(* Logix 5000 project; controller test vendor 1 type 14 code 196 rev 35.11; software revision 35.00 *)

TASK MainTask (continuous, watchdog 500 ms) : MainProgram

MODULES
   Local : vendor 1 type 14 code 196 (5069 0, rev 35.11)
END_MODULES

ADD_ON_INSTRUCTION Casting_Process   (* revision 1.0 *)
VAR_OUTPUT
   Header_Left : BOOL; {access Read Only, visible}
END_VAR
VAR_INPUT
   BW_Limit : BOOL; {required}
   Header_FW : BOOL; {required}
END_VAR
VAR_OUTPUT
   Casting : BOOL; {visible}
   Casting_Done : BOOL; {access Read Only, visible}
END_VAR
VAR
   Timer : TIMER := (PRE := 1500); {access None}
   Timer_1 : TIMER := (PRE := 2000); {access None}
END_VAR

ROUTINE Logic   (* ladder *)
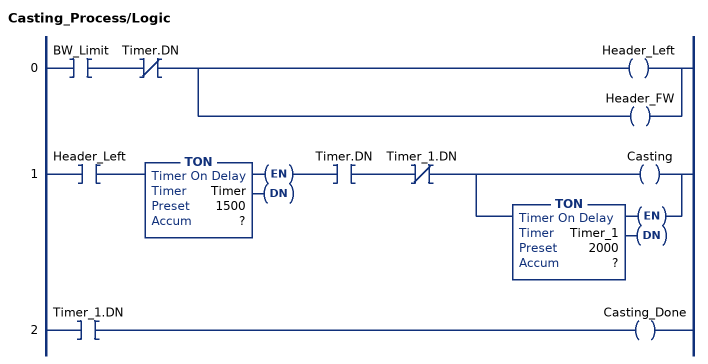
   0: XIC(BW_Limit)XIO(Timer.DN)[OTE(Header_Left) ,OTE(Header_FW) ];
   1: XIC(Header_Left)TON(Timer,?,?)XIC(Timer.DN)XIO(Timer_1.DN)[OTE(Casting) ,TON(Timer_1,?,?) ];
   2: XIC(Timer_1.DN)OTE(Casting_Done);
END_ROUTINE
END_ADD_ON_INSTRUCTION

ADD_ON_INSTRUCTION Molds_Tem   (* revision 1.0 *)
VAR_INPUT
   Temperature : REAL; {required}
END_VAR
VAR_OUTPUT
   Heating : BOOL; {access Read Only, visible}
   R : BOOL; {access Read Only, visible}
END_VAR

ROUTINE Logic   (* ladder *)
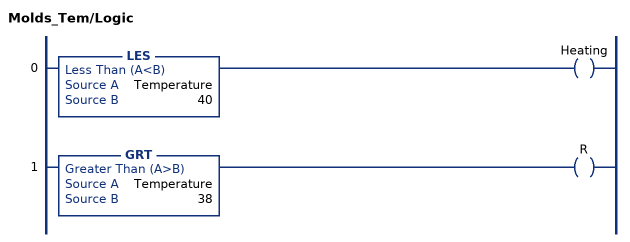
   0: LES(Temperature,40)OTE(Heating);
   1: GRT(Temperature,38)OTE(R);
END_ROUTINE
END_ADD_ON_INSTRUCTION

PROGRAM MainProgram   (* main routine MainRoutine *)
VAR
   Air_Valv : BOOL;
   BW_Limit : BOOL[32];
   Car_BW : BOOL;
   Car_Forward : BOOL;
   Car_FW : BOOL;
   Carriage : BOOL;
   Casting_Process_1 : Casting_Process;
   Casting_Process_2 : Casting_Process;
   Casting_Process_3 : Casting_Process;
   Casting_Process_4 : Casting_Process;
   Casting_Process_5 : Casting_Process;
   Casting_Process_6 : Casting_Process;
   Casting_Process_7 : Casting_Process;
   Casting_Process_8 : Casting_Process;
   Chem_Valv : BOOL;
   Emergency_Button : BOOL;
   Front_Limit : BOOL;
   FW_Limit : BOOL;
   Header_BW : BOOL;
   Header_FW : BOOL[32];
   Header_Right : BOOL;
   Initial_Position : BOOL;
   Light_Auto : BOOL;   // Automatic Light
   Light_Emer : BOOL;
   Light_Man : BOOL;   // Manual Light
   Manual : DINT;
   MTem_1 : Molds_Tem;
   MTem_2 : Molds_Tem;
   MTem_3 : Molds_Tem;
   MTem_4 : Molds_Tem;
   MTem_5 : Molds_Tem;
   MTem_6 : Molds_Tem;
   MTem_7 : Molds_Tem;
   MTem_8 : Molds_Tem;
   PB_AutoMan : BOOL;
   PB_Pouring_Material : BOOL;
   PB_Turn_Table : BOOL;
   PB_Valve_Air : BOOL;
   PB_Valve_Chemical : BOOL;
   Pouring_Material : BOOL;
   Preset_Time : DINT;
   Process_Auto : DINT;
   Process_Station : DINT;
   Ready : BOOL;
   Solenoid_with_chemical : BOOL;
   Solenoid_with_compressed_air : BOOL;
   Start_Button : BOOL;
   Strain : BOOL;
   Switch_Car_BW : BOOL;
   Switch_Car_Forward : BOOL;
   Switch_Header_BW : BOOL;
   Switch_Header_FW : BOOL;
   Tem_1 : REAL;
   Tem_2 : REAL;
   Tem_3 : REAL;
   Tem_4 : REAL;
   Tem_5 : REAL;
   Tem_6 : REAL;
   Tem_7 : REAL;
   Tem_8 : REAL;
   Tem_Ready : BOOL;
   Time_Air_Valv : TIMER := (PRE := 3000);
   Time_Chem_Valv : TIMER := (PRE := 1000);
   Time_Strain : DINT;
   Timer_1 : TIMER := (PRE := 10000);
   Timer_2 : TIMER := (PRE := 1500);
   Turn_Table : BOOL;
END_VAR

ROUTINE Automatic   (* ladder *)
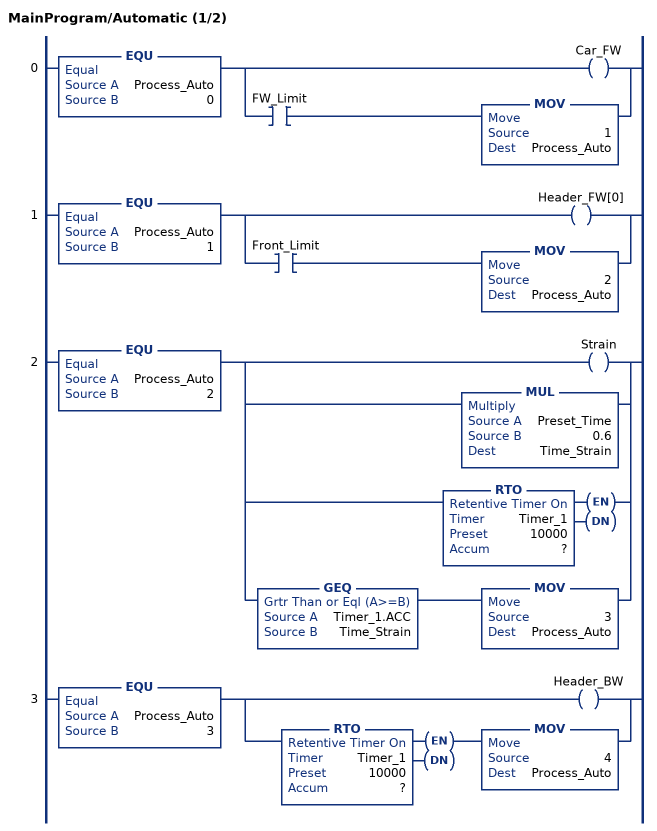
   0: EQU(Process_Auto,0)[OTE(Car_FW) ,XIC(FW_Limit) MOV(1,Process_Auto) ];
   1: EQU(Process_Auto,1)[OTE(Header_FW[0]) ,XIC(Front_Limit) MOV(2,Process_Auto) ];
   2: EQU(Process_Auto,2)[[OTE(Strain) ,MUL(Preset_Time,0.6,Time_Strain) ,RTO(Timer_1,?,?) ] ,GEQ(Timer_1.ACC,Time_Strain) MOV(3,Process_Auto) ];
   3: EQU(Process_Auto,3)[OTE(Header_BW) ,RTO(Timer_1,?,?) MOV(4,Process_Auto) ];
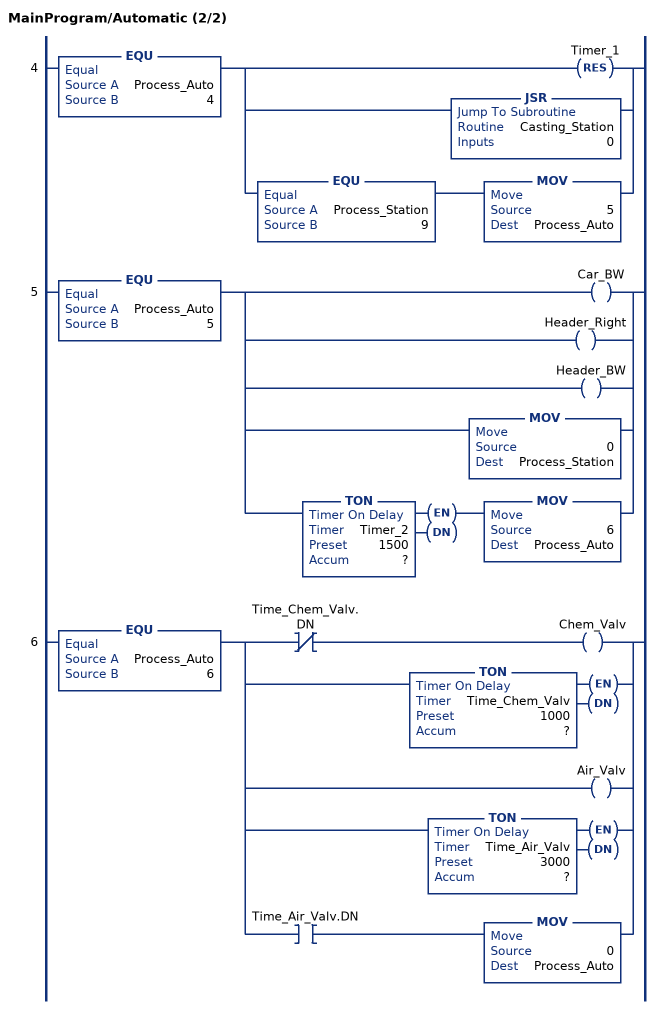
   4: EQU(Process_Auto,4)[[RES(Timer_1) ,JSR(Casting_Station,0) ] ,EQU(Process_Station,9) MOV(5,Process_Auto) ];
   5: EQU(Process_Auto,5)[[[OTE(Car_BW) ,OTE(Header_Right) ,OTE(Header_BW) ] ,MOV(0,Process_Station) ] ,TON(Timer_2,?,?) MOV(6,Process_Auto) ];
   6: EQU(Process_Auto,6)[[[XIO(Time_Chem_Valv.DN) OTE(Chem_Valv) ,TON(Time_Chem_Valv,?,?) ] ,[OTE(Air_Valv) ,TON(Time_Air_Valv,?,?) ] ] ,XIC(Time_Air_Valv.DN) MOV(0,Process_Auto) ];
END_ROUTINE

ROUTINE Casting_Station   (* ladder *)
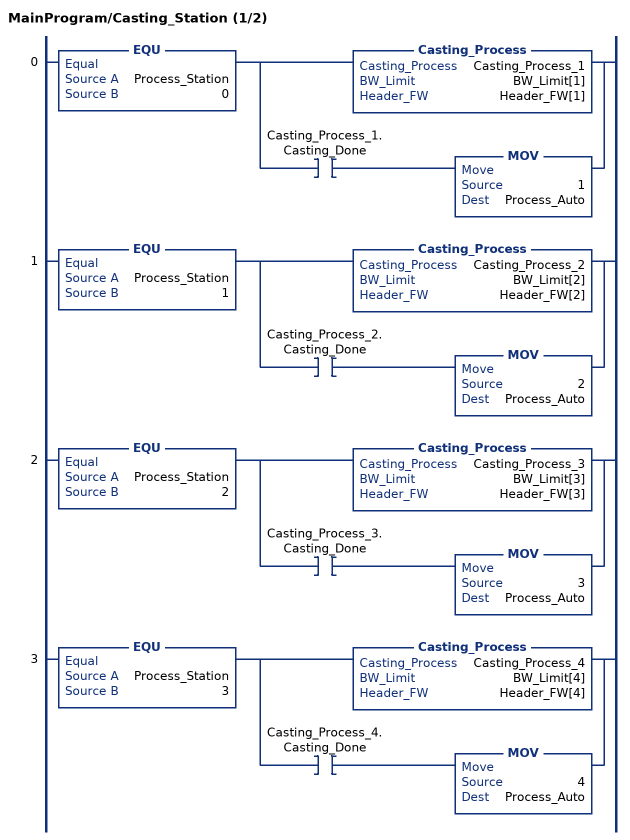
   0: EQU(Process_Station,0)[Casting_Process(Casting_Process_1,BW_Limit[1],Header_FW[1]) ,XIC(Casting_Process_1.Casting_Done) MOV(1,Process_Auto) ];
   1: EQU(Process_Station,1)[Casting_Process(Casting_Process_2,BW_Limit[2],Header_FW[2]) ,XIC(Casting_Process_2.Casting_Done) MOV(2,Process_Auto) ];
   2: EQU(Process_Station,2)[Casting_Process(Casting_Process_3,BW_Limit[3],Header_FW[3]) ,XIC(Casting_Process_3.Casting_Done) MOV(3,Process_Auto) ];
   3: EQU(Process_Station,3)[Casting_Process(Casting_Process_4,BW_Limit[4],Header_FW[4]) ,XIC(Casting_Process_4.Casting_Done) MOV(4,Process_Auto) ];
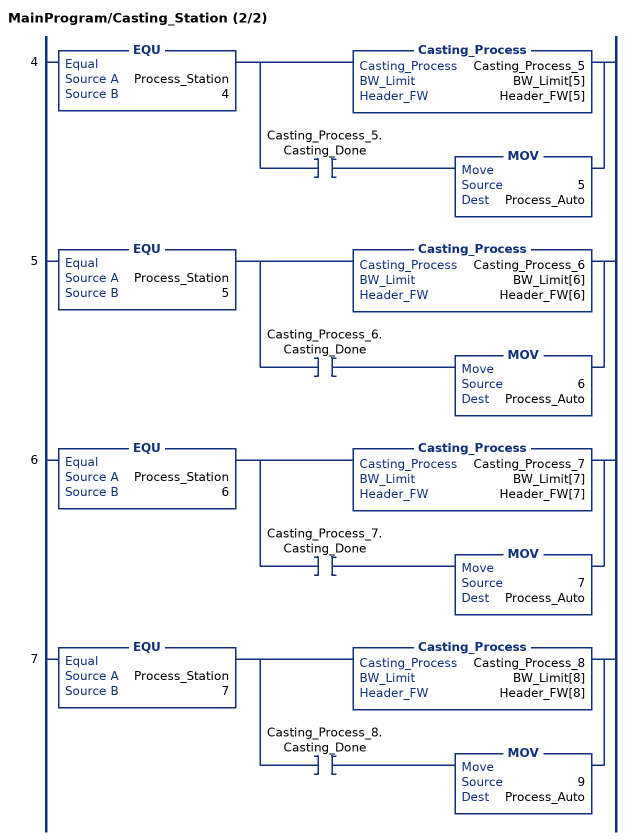
   4: EQU(Process_Station,4)[Casting_Process(Casting_Process_5,BW_Limit[5],Header_FW[5]) ,XIC(Casting_Process_5.Casting_Done) MOV(5,Process_Auto) ];
   5: EQU(Process_Station,5)[Casting_Process(Casting_Process_6,BW_Limit[6],Header_FW[6]) ,XIC(Casting_Process_6.Casting_Done) MOV(6,Process_Auto) ];
   6: EQU(Process_Station,6)[Casting_Process(Casting_Process_7,BW_Limit[7],Header_FW[7]) ,XIC(Casting_Process_7.Casting_Done) MOV(7,Process_Auto) ];
   7: EQU(Process_Station,7)[Casting_Process(Casting_Process_8,BW_Limit[8],Header_FW[8]) ,XIC(Casting_Process_8.Casting_Done) MOV(9,Process_Auto) ];
END_ROUTINE

ROUTINE MainRoutine   (* ladder *)
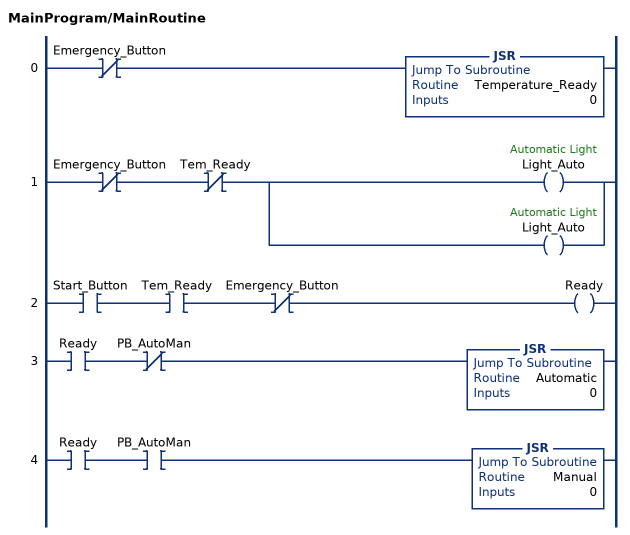
   0: XIO(Emergency_Button)JSR(Temperature_Ready,0);
   1: XIO(Emergency_Button)XIO(Tem_Ready)[OTE(Light_Auto) ,OTE(Light_Auto) ];
   2: XIC(Start_Button)XIC(Tem_Ready)XIO(Emergency_Button)OTE(Ready);
   3: XIC(Ready)XIO(PB_AutoMan)JSR(Automatic,0);
   4: XIC(Ready)XIC(PB_AutoMan)JSR(Manual,0);
END_ROUTINE

ROUTINE Manual   (* ladder *)
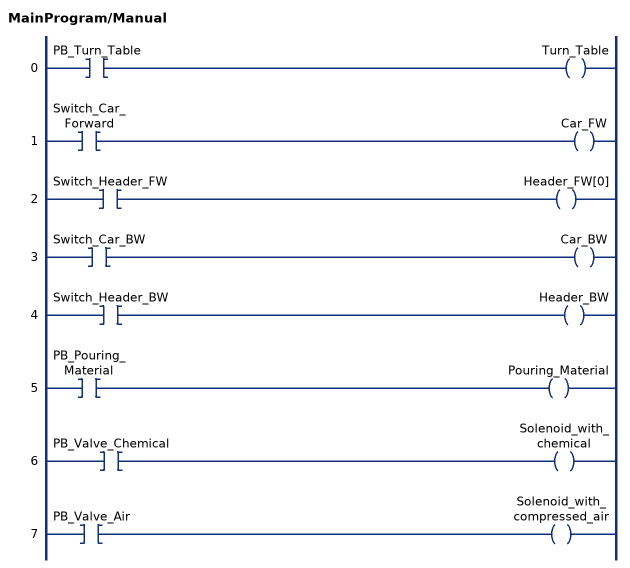
   0: XIC(PB_Turn_Table)OTE(Turn_Table);
   1: XIC(Switch_Car_Forward)OTE(Car_FW);
   2: XIC(Switch_Header_FW)OTE(Header_FW[0]);
   3: XIC(Switch_Car_BW)OTE(Car_BW);
   4: XIC(Switch_Header_BW)OTE(Header_BW);
   5: XIC(PB_Pouring_Material)OTE(Pouring_Material);
   6: XIC(PB_Valve_Chemical)OTE(Solenoid_with_chemical);
   7: XIC(PB_Valve_Air)OTE(Solenoid_with_compressed_air);
END_ROUTINE

ROUTINE Temperature_Ready   (* ladder *)
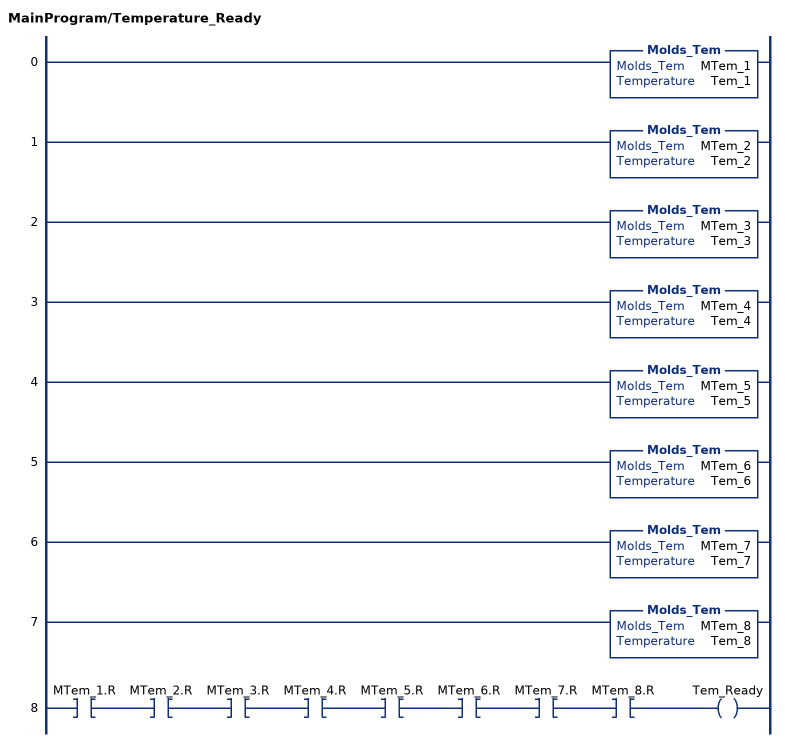
   0: Molds_Tem(MTem_1,Tem_1);
   1: Molds_Tem(MTem_2,Tem_2);
   2: Molds_Tem(MTem_3,Tem_3);
   3: Molds_Tem(MTem_4,Tem_4);
   4: Molds_Tem(MTem_5,Tem_5);
   5: Molds_Tem(MTem_6,Tem_6);
   6: Molds_Tem(MTem_7,Tem_7);
   7: Molds_Tem(MTem_8,Tem_8);
   8: XIC(MTem_1.R)XIC(MTem_2.R)XIC(MTem_3.R)XIC(MTem_4.R)XIC(MTem_5.R)XIC(MTem_6.R)XIC(MTem_7.R)XIC(MTem_8.R)OTE(Tem_Ready);
END_ROUTINE
END_PROGRAM
